{attribute 'OPC.UA.DA' := '1'}
{attribute 'OPC.UA.DA.StructuredType' := '1'}
TYPE IdentifierMsg :
STRUCT
	Id : EPowerIlluminationFlow;
	Identifier : STRING(255);
END_STRUCT
END_TYPE

(* stored: Version 1.1.0.1, ProductVersion 3.1.4024.3
   DUT IdentifierMsg: Id {3b94029f-fde8-43a6-934f-f13f3f89bbae} *)
